// TwinCAT 3 PLC project ZK_Doc1
// Title: Doc-Test
// Company: Lisec
// Author: reschsim
// ProjectVersion: 0.4.0
// ProgramVersion: 3.1.4026.25
// libraries:
//   Tc2_Standard, * (Beckhoff Automation GmbH)
//   Tc2_System, * (Beckhoff Automation GmbH)
// project tree:
//   DUTs/ DUT.TcTLEO, ST_Base.TcDUT, ST_Test1.TcDUT
//   GVLs/ GVL_Test1.TcGVL
//   ITFs/ I_Base.TcIO
//   POUs/ FB_Test1_Base.TcPOU, F_Test1.TcPOU, POU.TcPOU, FB_Test1.TcPOU
//   Project Information/ F_GetCompany.TcPOU, F_GetTitle.TcPOU, F_GetVersion.TcPOU
//   Version/ Global_Version.TcGVL
// real-time tasks:
//   TASK PlcTask: cycle T#10ms, priority 20, ADS port 350
//   TASK PlcTask1: cycle T#10ms, priority 21, ADS port 351

// ---- DUTs/DUT.TcTLEO
{attribute 'qualified_only'}
{attribute 'strict'}
{attribute 'to_string'}
/// Enum ***DUT***
TYPE DUT :
(
	member1 := 0, //< default
	member2 := 10, //< nr 10
	meber3 := 20, //< nr 20
	meber4 := 30 //< nr 30
);
END_TYPE
//  meber4 = '30 '

// ---- DUTs/ST_Base.TcDUT
/// the base struct for every coming struct
/// ---
/// now a Table
///| Syntax      | Description | Test Text     |
///| :---        |    :----:   |          ---: |
///| Header      | Title       | Here's this   |
///| Paragraph   | Text        | And more      |
TYPE ST_Base :
STRUCT
	nTest1 : INT; //< for testing
	nTest2 : INT; //< also for testing
	nTest3 : INT; //< just for *testing*
END_STRUCT
END_TYPE

// ---- DUTs/ST_Test1.TcDUT
TYPE ST_Test1 EXTENDS ST_Base :
STRUCT
	nTest4 : INT;
	stBase : ST_Base;
END_STRUCT
END_TYPE

// ---- GVLs/GVL_Test1.TcGVL
{attribute 'qualified_only'}
/// This is a Test **GVL**
VAR_GLOBAL //< now comes the variables
	nGVar1 : INT;
	aGVar2 : ARRAY[0..100] OF INT;
END_VAR
VAR_GLOBAL PERSISTENT
	nPersGVar1 : INT; //< this is a persistent var
END_VAR
VAR_GLOBAL CONSTANT
	nConst1 : INT := 1; //< for constant use
	nConst2 : INT := 2;
	nConst3 : INT := 3; //< for constant use
	nConst4 : INT := 4;
END_VAR

// ---- Version/Global_Version.TcGVL
{attribute 'TcGenerated'}
{attribute 'no-analysis'}
{attribute 'linkalways'}
// This function has been automatically generated from the project information.
VAR_GLOBAL CONSTANT
	{attribute 'const_non_replaced'}
	stLibVersion_Doc_Test : ST_LibVersion := (iMajor := 0, iMinor := 4, iBuild := 0, iRevision := 0, nFlags := 0, sVersion := '0.4.0');
END_VAR

// ---- ITFs/I_Base.TcIO
INTERFACE I_Base

/// This is a TestMethod
METHOD M_Test1 : INT
VAR_INPUT
END_VAR
END_METHOD

/// A Test Property with get and set
PROPERTY P_TestFor : BOOL
GET
END_GET
SET
END_SET
END_PROPERTY

END_INTERFACE

// ---- POUs/FB_Test1_Base.TcPOU
/// This is the **Base** FB for every single FB
/// Inherited by:
FUNCTION_BLOCK FB_Test1_Base //< [FB_Test1](xref:ZK_Doc1.FB_Test1)
VAR_INPUT
	/// This is the first ___Input___
	/// Now comes a code example:
	/// ~~We dont need this~~
	/// ```st
	/// METHOD Method1
	/// VAR_INPUT
  	/// input1 : BOOL; //< what does this input do
  	///
  	/// /// or this one?
  	/// input2 : INT;
	/// END_VAR
	/// ```
	nInput1 : INT := 1; 
END_VAR
VAR_OUTPUT
	sOutput1 : T_MaxString := "This is output 1";
END_VAR
VAR
	nVar1 : INT;
	nVar2 : INT;
	sVar3 : T_MaxString;
	bVar4 : BOOL;
END_VAR
VAR CONSTANT
	nConst1 : INT := 2026;
	sConst2 : STRING(155) := 'Constant 2';
END_VAR
VAR PERSISTENT
	nVarPers : LREAL := 155.155;
	
END_VAR

METHOD INTERNAL M_SetVar : BOOL
VAR_INPUT
	nVarIn1 : INT;
END_VAR
P_nVar1 := nVarIn1;
M_SetVar := nVarIn1 >= 100;
RETURN;
END_METHOD

PROPERTY PRIVATE P_FOO : BOOL
GET
P_FOO := TRUE;
RETURN;
END_GET
SET
bVar4 := P_FOO;
END_SET
END_PROPERTY

PROPERTY PROTECTED P_nVar1 : INT
GET
P_nVar1 := nVar1;
RETURN;
END_GET
SET
nVar1 := P_nVar1;
END_SET
END_PROPERTY

END_FUNCTION_BLOCK

// ---- POUs/F_Test1.TcPOU
/// here comes a function (**FUN**)
/// ---
/// And now a mermaid.js diagramm
/// ```mermaid
///	stateDiagram-v2
/// 	[*] --> Init: PLC started
///		Init --> GoHome: home pressed
/// 	GoHome --> Idle: done
///		GoHome --> FaultReaction: aborted
/// 	FaultReaction --> Init: done\nnot initialized
///		FaultReaction --> Idle: done
///		Idle --> GoHome: home pressed
///	```
FUNCTION F_Test1 : BOOL
VAR_INPUT
	stInput : ST_Test1; //< input1
END_VAR
VAR
END_VAR

F_Test1 := stInput.stBase.nTest1 < 100;
RETURN;

END_FUNCTION

// ---- POUs/POU.TcPOU
/// Link to Lisec [Lisec](https://www.lisec.com)
///![Lisec](./../documentation/images/logo.png)
/// This a empty **POU**
PROGRAM POU
VAR
	i : INT;
END_VAR

i;

METHOD ABSTRACT M_Test1 : BOOL
VAR_INPUT
	sTest1 : T_MaxString;
	nTest2 : LREAL;
END_VAR
END_METHOD

PROPERTY PROTECTED ABSTRACT P_BAR : BOOL
END_PROPERTY

END_PROGRAM

// ---- POUs/FB_Test1.TcPOU
FUNCTION_BLOCK FB_Test1 EXTENDS FB_Test1_Base IMPLEMENTS I_Base
VAR_INPUT
END_VAR
VAR_OUTPUT
END_VAR
VAR
END_VAR

{warning 'Methodenimplementierung hinzufügen'}
METHOD M_Test1 : INT
END_METHOD

{warning 'Eigenschaftenimplementierung hinzufügen'}
PROPERTY P_TestFor : BOOL
GET
END_GET
SET
END_SET
END_PROPERTY

END_FUNCTION_BLOCK

// ---- Project Information/F_GetCompany.TcPOU
// This function has been automatically generated from the project information.
{attribute 'signature_flag' := '1073741824'}
{attribute 'TcGenerated'}
{attribute 'no-analysis'}
FUNCTION F_GetCompany : WSTRING
VAR_INPUT
	
END_VAR

F_GetCompany := "Lisec";

END_FUNCTION

// ---- Project Information/F_GetTitle.TcPOU
// This function has been automatically generated from the project information.
{attribute 'signature_flag' := '1073741824'}
{attribute 'TcGenerated'}
{attribute 'no-analysis'}
FUNCTION F_GetTitle : WSTRING
VAR_INPUT
	
END_VAR

F_GetTitle := "Doc-Test";

END_FUNCTION

// ---- Project Information/F_GetVersion.TcPOU
// This function has been automatically generated from the project information.
{attribute 'signature_flag' := '1073741824'}
{attribute 'TcGenerated'}
{attribute 'no-analysis'}
FUNCTION F_GetVersion : ST_LibVersion
VAR_INPUT
	
END_VAR

F_GetVersion.iMajor := 0;
F_GetVersion.iMinor := 4;
F_GetVersion.iBuild := 0;
F_GetVersion.iRevision := 0;
F_GetVersion.sVersion := '0.4.0';
F_GetVersion.nFlags := 0;

END_FUNCTION
